// TIA Portal V16 export
// export: Created 2022-07-21T09:35:18.3308765Z, ExportSetting WithDefaults, DisplayName Totally Integrated Automation Portal, DisplayVersion V16 Update 4, DisplayName TIA Portal Version Control Interface, DisplayVersion V16 Update 2, DisplayName TIA Portal Openness, DisplayVersion V16 Update 4, DisplayName SINAMICS Startdrive Advanced, DisplayVersion V16 Update 5, DisplayName SINAMICS Startdrive G130, G150, S120, S150, SINAMICS MV, S210, DisplayVersion V16 Update 5, DisplayName SINAMICS Startdrive G110M, G120, G120C, G120D, G120P, G115D, DisplayVersion V16 Update 5, DisplayName STEP 7 Professional, DisplayVersion V16 Update 4, DisplayName STEP 7 Safety, DisplayVersion V16, DisplayName WinCC Advanced, DisplayVersion V16 Update 4
FUNCTION_BLOCK "fbATI"   // FB20, LAD
TITLE = ATI / Blok do obsługi ATI
{ S7_Optimized_Access := 'TRUE' }
VERSION : 0.1
// stored: AutoNumber false, IsIECCheckEnabled false, IsRetainMemResEnabled false, MemoryReserve 100, SetENOAutomatically false, UDAEnableTagReadback false
   VAR_INPUT
      portNr : UInt;   // numer portu / Port number
      generalRelease { ExternalWritable := 'False'} : Bool;   // Zezwolenie / General release
      autoEnable { ExternalWritable := 'False'} : Bool := true;   // Tryb automatyczny z HMI / Automatic mode from HMI
      ATI_ready { ExternalWritable := 'False'} : Bool;   // ATI -> PLC gotowe / ATI -> PLC ready
      ATI_passedTst { ExternalWritable := 'False'} : Bool;   // ATI -> PLC test ok
      ATI_failedTst { ExternalWritable := 'False'} : Bool;   // ATI -> PLC test nok
      ATI_fault { ExternalWritable := 'False'} : Bool;   // ATI -> PLC błąd / ATI -> PLC fault
      ATI_calMode { ExternalWritable := 'False'} : Bool;   // ATI -> PLC tryb kalibracji / ATI -> PLC calibration
      chuckClosed { ExternalWritable := 'False'} : Bool;   // Chuck zamknięty / Chuck closed
      partPlaced { ExternalWritable := 'False'} : Bool;   // Filtr w pozycji / Filter in position
      autoPenCal : Bool;   // Żądanie kalibracji / Calibration request
      group : "typeGroup";   // Grupa / Group
   END_VAR
   VAR_OUTPUT
      autoSelect { ExternalWritable := 'False'} : Bool;   // PLC -> ATI Tryb auto / PLC -> ATI Automatic mode
      extStart { ExternalWritable := 'False'} : Bool;   // PLC -> ATI Zewnętrzny start / PLC -> ATI External start
      penCal { ExternalWritable := 'False'} : Bool;   // PLC -> ATI Pen Cal
      ATIexists { ExternalWritable := 'False'} : Bool;   // ATI -> ext. ATI załączone z HMI / ATI -> ext. ATI on from HMI
      calIsRunning : Bool;   // kalibracja aktywna / calibration active
      calElapsedTime : Time;   // czas trwania kalibracji / calibration duration
      errorSendPort : Bool;   // Błąd bloku P2P Send / Block error P2P Send
      errorRecvPort : Bool;   // Błąd bloku P2P Receive / Block error P2P Receive
      errorCom : Bool;   // Błąd koumikacji : związany z Receive / Communication error : Receive related
   END_VAR
   VAR_IN_OUT
      ATI : "typeTester";   // Dane HMI / HMI data
      ATIP2P : "typeATIP2P";
      instRecvP2P : Receive_P2P;
      instSendP2P : Send_P2P;
   END_VAR
   VAR
      statTimerPenCalPls { ExternalWritable := 'False'; S7_SetPoint := 'True'} : TON_TIME;
      statTimerStartPls { ExternalWritable := 'False'; S7_SetPoint := 'True'} : TON_TIME;
      staRecvNDR { S7_SetPoint := 'True'} : Bool;
      statRecvError : Bool;
      statRecvStatus : Word;
      statRecvLength : UInt;
      statRecievedData : String;
      statSendData : String;
      statSendTrigger : Bool;
      statSendLength : UInt;
      statSendDone : Bool;
      statSendError : Bool;
      statSendStatus : Word;
      stat1Char : String;
      instDelaySendTG : TP_TIME;
      instDelayErrorRecvTG : TON_TIME;
      statWaitingForRecvTG : Bool;
      statDelayErrorProcess : Time;
      NewResultOKDigit { S7_SetPoint := 'True'} : Bool;
      NewResultOKDigit_RTIG : R_TRIG;
      NewResultNOKDigit : Bool;
      NewResultNOKDigit_RTIG : R_TRIG;
      sNegEdge : Array[0..7] of Bool;
      sPosEdge : Array[0..7] of Bool;
      sEqual : Bool;
   END_VAR
   VAR_TEMP
      tempCancelCalMode : Bool;   // Reset trybu kalibracji / Reset calibration mode
      tempAutoModeActive : Bool;   // Tryb auto/krokowy aktywny / Automatic/sequential mode active
      tempModeActive : Bool;   // Tryb aktywny / Active mode
      tempRetVal : Int;
      tempREQSend : Bool;
      tempCount : Int;
      tempVarTimeCAL : Time;
      tempCALerror : Bool;
      temp_cRL : Char;
      temp_sRL : String;
      tempStr : String;
      tempEqual : Bool;
      tempStatus3 : Bool;
   END_VAR
   VAR CONSTANT
      cTIME_OFF_SIGNAL : Time := T#1s;   // Czas opóźnienia dla alarmu 0 / delay alarm 0
      cTIME_ERR_PROCESS : Time := T#90s;
   END_VAR
   // // ATI.cmd.enable : Włączenie trybu automatycznego / Start automatic mode
   VAR_TEMP   // added for the SCL form of the ladder/FBD networks
      _w1 : Bool;
      _w2 : Bool;
   END_VAR
BEGIN

REGION Network 1: Alarm 1 - ATI fault / Alarm 1 - Błąd ATI
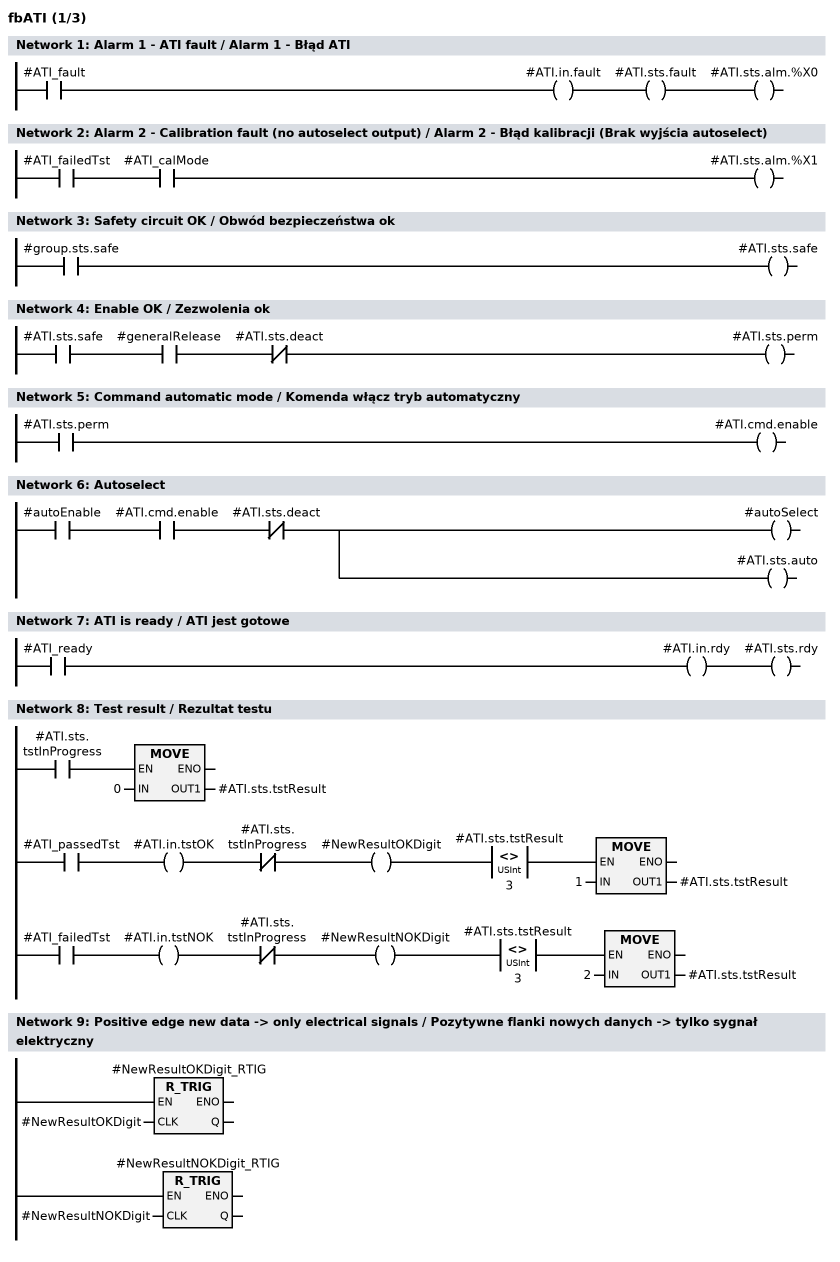
   RUNG wire#powerrail
      Contact( #ATI_fault )
      Coil( #ATI.in.fault )
      Coil( #ATI.sts.fault )
      Coil( #ATI.sts.alm.%X0 )
   END_RUNG
   // the same network as SCL:
   #ATI.in.fault := #ATI_fault;
   #ATI.sts.fault := #ATI_fault;
   #ATI.sts.alm.%X0 := #ATI_fault;
END_REGION

REGION Network 2: Alarm 2 - Calibration fault (no autoselect output) / Alarm 2 - Błąd kalibracji (Brak wyjścia autoselect)
   RUNG wire#powerrail
      Contact( #ATI_failedTst )
      Contact( #ATI_calMode )
      Coil( #ATI.sts.alm.%X1 )
   END_RUNG
   // the same network as SCL:
   #ATI.sts.alm.%X1 := #ATI_failedTst AND #ATI_calMode;
END_REGION

REGION Network 3: Safety circuit OK / Obwód bezpieczeństwa ok
   RUNG wire#powerrail
      Contact( #group.sts.safe )
      Coil( #ATI.sts.safe )
   END_RUNG
   // the same network as SCL:
   #ATI.sts.safe := #group.sts.safe;
END_REGION

REGION Network 4: Enable OK / Zezwolenia ok
   RUNG wire#powerrail
      Contact( #ATI.sts.safe )
      Contact( #generalRelease )
      I_Contact( #ATI.sts.deact )
      Coil( #ATI.sts.perm )
   END_RUNG
   // the same network as SCL:
   #ATI.sts.perm := #ATI.sts.safe AND #generalRelease AND NOT #ATI.sts.deact;
END_REGION

REGION Network 5: Command automatic mode / Komenda włącz tryb automatyczny
   RUNG wire#powerrail
      Contact( #ATI.sts.perm )
      Coil( #ATI.cmd.enable )
   END_RUNG
   // the same network as SCL:
   #ATI.cmd.enable := #ATI.sts.perm;
END_REGION

REGION Network 6: Autoselect
   RUNG wire#powerrail
      Contact( #autoEnable )
      Contact( #ATI.cmd.enable )
      I_Contact( #ATI.sts.deact )
      wire#w1
      Coil( #autoSelect )
   END_RUNG
   RUNG wire#w1
      Coil( #ATI.sts.auto )
   END_RUNG
   // the same network as SCL:
   #autoSelect := #autoEnable AND #ATI.cmd.enable AND NOT #ATI.sts.deact;
   #ATI.sts.auto := #autoSelect;
END_REGION

REGION Network 7: ATI is ready / ATI jest gotowe
   RUNG wire#powerrail
      Contact( #ATI_ready )
      Coil( #ATI.in.rdy )
      Coil( #ATI.sts.rdy )
   END_RUNG
   // the same network as SCL:
   #ATI.in.rdy := #ATI_ready;
   #ATI.sts.rdy := #ATI_ready;
END_REGION

REGION Network 8: Test result / Rezultat testu
   RUNG wire#powerrail
      Contact( #ATI.sts.tstInProgress )
      Move(in := 0, out1 => #ATI.sts.tstResult)
   END_RUNG
   RUNG wire#powerrail
      Contact( #ATI_passedTst )
      Coil( #ATI.in.tstOK )
      I_Contact( #ATI.sts.tstInProgress )
      Coil( #NewResultOKDigit )
      { S7_Templates := "SrcType := USInt" } NE_Contact(in1 := #ATI.sts.tstResult, in2 := 3)
      Move(in := 1, out1 => #ATI.sts.tstResult)
   END_RUNG
   RUNG wire#powerrail
      Contact( #ATI_failedTst )
      Coil( #ATI.in.tstNOK )
      I_Contact( #ATI.sts.tstInProgress )
      Coil( #NewResultNOKDigit )
      { S7_Templates := "SrcType := USInt" } NE_Contact(in1 := #ATI.sts.tstResult, in2 := 3)
      Move(in := 2, out1 => #ATI.sts.tstResult)
   END_RUNG
   // the same network as SCL:
   IF #ATI.sts.tstInProgress THEN #ATI.sts.tstResult := 0; END_IF;
   #ATI.in.tstOK := #ATI_passedTst;
   #NewResultOKDigit := #ATI_passedTst AND NOT #ATI.sts.tstInProgress;
   IF #NewResultOKDigit AND (#ATI.sts.tstResult <> 3) THEN #ATI.sts.tstResult := 1; END_IF;
   #ATI.in.tstNOK := #ATI_failedTst;
   #NewResultNOKDigit := #ATI_failedTst AND NOT #ATI.sts.tstInProgress;
   IF #NewResultNOKDigit AND (#ATI.sts.tstResult <> 3) THEN #ATI.sts.tstResult := 2; END_IF;
END_REGION

REGION Network 9: Positive edge new data -> only electrical signals / Pozytywne flanki nowych danych -> tylko sygnał elektryczny
   RUNG wire#powerrail
      #NewResultOKDigit_RTIG.R_TRIG(CLK := #NewResultOKDigit, Q =>)
   END_RUNG
   RUNG wire#powerrail
      #NewResultNOKDigit_RTIG.R_TRIG(CLK := #NewResultNOKDigit, Q =>)
   END_RUNG
   // the same network as SCL:
   #NewResultOKDigit_RTIG(CLK := #NewResultOKDigit);   // R_TRIG
   #NewResultNOKDigit_RTIG(CLK := #NewResultNOKDigit);   // R_TRIG
END_REGION

REGION Network 10: Alarm 4 - No RS232 data after test / Alarm 4 - Brak danych RS232 po teście
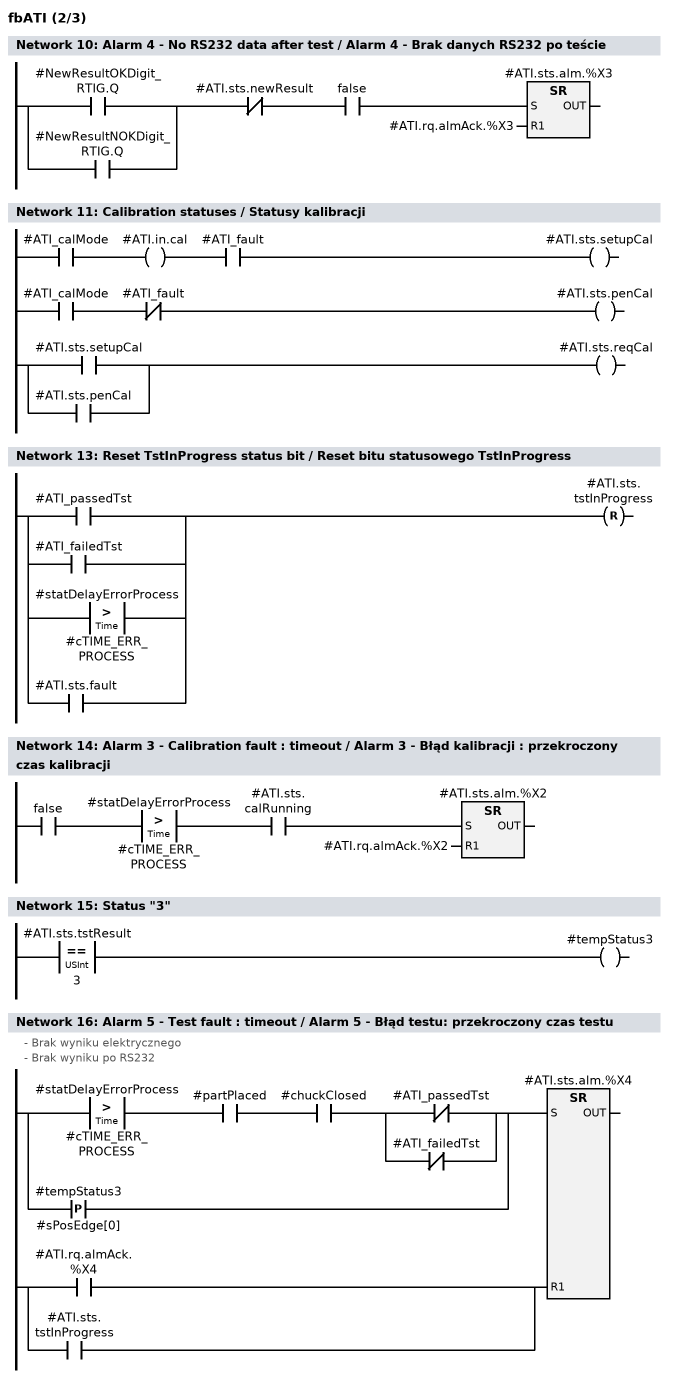
   RUNG wire#powerrail
      Contact( #NewResultOKDigit_RTIG.Q )
      wire#w1
      I_Contact( #ATI.sts.newResult )
      Contact( false )
      S_SR(operand := #ATI.sts.alm.%X3, r1 := #ATI.rq.almAck.%X3)
   END_RUNG
   RUNG wire#powerrail
      Contact( #NewResultNOKDigit_RTIG.Q )
   END_RUNG wire#w1
   // the same network as SCL:
   IF (#NewResultOKDigit_RTIG.Q OR #NewResultNOKDigit_RTIG.Q) AND NOT #ATI.sts.newResult AND false THEN
       #ATI.sts.alm.%X3 := TRUE;   // SR flip-flop
   END_IF;
   IF #ATI.rq.almAck.%X3 THEN #ATI.sts.alm.%X3 := FALSE; END_IF;
END_REGION

REGION Network 11: Calibration statuses / Statusy kalibracji
   RUNG wire#powerrail
      Contact( #ATI_calMode )
      Coil( #ATI.in.cal )
      Contact( #ATI_fault )
      Coil( #ATI.sts.setupCal )
   END_RUNG
   RUNG wire#powerrail
      Contact( #ATI_calMode )
      I_Contact( #ATI_fault )
      Coil( #ATI.sts.penCal )
   END_RUNG
   RUNG wire#powerrail
      Contact( #ATI.sts.setupCal )
      wire#w1
      Coil( #ATI.sts.reqCal )
   END_RUNG
   RUNG wire#powerrail
      Contact( #ATI.sts.penCal )
   END_RUNG wire#w1
   // the same network as SCL:
   #ATI.in.cal := #ATI_calMode;
   #ATI.sts.setupCal := #ATI_calMode AND #ATI_fault;
   #ATI.sts.penCal := #ATI_calMode AND NOT #ATI_fault;
   #ATI.sts.reqCal := #ATI.sts.setupCal OR #ATI.sts.penCal;
END_REGION

REGION Network 12 (SCL): ATI control / Sterowanie ATI

   #tempAutoModeActive := #group.sts.auto OR #group.sts.step;
   #tempModeActive := #tempAutoModeActive OR #group.sts.manual; //jakikolwiek tryb wybrany

   //Testy filtrów
   IF #ATI_ready AND NOT #ATI_fault THEN

       //start test filtra
       IF #autoSelect AND ((#tempAutoModeActive AND #partPlaced) OR (#group.sts.manual AND #ATI.rq.handStart))
           AND #chuckClosed AND NOT (#ATI_passedTst OR #ATI_failedTst) AND NOT #extStart THEN
           #extStart := TRUE;
           #ATI.sts.tstInProgress := TRUE;
       END_IF;

       //wymuszenie kalibracji podczas normalnej pracy
       IF #autoSelect AND #group.sts.manual AND NOT #partPlaced AND #chuckClosed AND #ATI.rq.rqPenCal AND NOT #penCal THEN
           #penCal := TRUE;
       END_IF;

   //Zadanie kalibracji
   ELSIF #ATI_calMode THEN

       //po starcie systemu (bład na ATI)
       IF #ATI.sts.setupCal THEN

           //tylko w trybie recznym ?
           IF #group.sts.manual AND #autoSelect AND NOT #partPlaced AND #chuckClosed AND #ATI.rq.startCal AND NOT #extStart THEN
               #extStart := TRUE;
               #ATI.sts.calRunning := TRUE;
           END_IF;

       //podczas normalnej pracy, po wcześniejszym jego wymuszeniu    
       ELSIF #ATI.sts.penCal THEN

           IF #tempModeActive AND #autoSelect AND NOT #partPlaced AND #chuckClosed AND (#ATI.rq.startCal OR #autoPenCal) AND NOT #extStart THEN
               #extStart := TRUE;
               #ATI.sts.calRunning := TRUE;
           END_IF;
       END_IF;
   END_IF;

   #statTimerStartPls(IN := #extStart,
                      PT := #cTIME_OFF_SIGNAL);
   #statTimerPenCalPls(IN := #penCal,
                       PT := #cTIME_OFF_SIGNAL);

   "fcCounterTime"(inEnableCount := true,
                   inReset := #extStart,
                   inValue := "CycleTimeData".PrevScanTime.Time,
                   ioCounter := #statDelayErrorProcess);

   IF #statTimerStartPls.Q THEN
       #extStart := FALSE;
   END_IF;

   IF #statTimerPenCalPls.Q THEN
       #penCal := FALSE;
   END_IF;

   IF #ATI.sts.calRunning THEN
       #calIsRunning := TRUE;
       #calElapsedTime := #statDelayErrorProcess;
   ELSE
       #calIsRunning := FALSE;
       #calElapsedTime := t#0ms;
   END_IF;
END_REGION

REGION Network 13: Reset TstInProgress status bit / Reset bitu statusowego TstInProgress
   RUNG wire#powerrail
      Contact( #ATI_passedTst )
      wire#w1
      R_Coil( #ATI.sts.tstInProgress )
   END_RUNG
   RUNG wire#powerrail
      Contact( #ATI_failedTst )
   END_RUNG wire#w1
   RUNG wire#powerrail
      { S7_Templates := "SrcType := Time" } GT_Contact(in1 := #statDelayErrorProcess, in2 := #cTIME_ERR_PROCESS)
   END_RUNG wire#w1
   RUNG wire#powerrail
      Contact( #ATI.sts.fault )
   END_RUNG wire#w1
   // the same network as SCL:
   IF #ATI_passedTst OR #ATI_failedTst OR (#statDelayErrorProcess > #cTIME_ERR_PROCESS) OR #ATI.sts.fault THEN
       #ATI.sts.tstInProgress := FALSE;
   END_IF;
END_REGION

REGION Network 14: Alarm 3 - Calibration fault : timeout / Alarm 3 - Błąd kalibracji : przekroczony czas kalibracji
   RUNG wire#powerrail
      Contact( false )
      { S7_Templates := "SrcType := Time" } GT_Contact(in1 := #statDelayErrorProcess, in2 := #cTIME_ERR_PROCESS)
      Contact( #ATI.sts.calRunning )
      S_SR(operand := #ATI.sts.alm.%X2, r1 := #ATI.rq.almAck.%X2)
   END_RUNG
   // the same network as SCL:
   IF false AND (#statDelayErrorProcess > #cTIME_ERR_PROCESS) AND #ATI.sts.calRunning THEN
       #ATI.sts.alm.%X2 := TRUE;   // SR flip-flop
   END_IF;
   IF #ATI.rq.almAck.%X2 THEN #ATI.sts.alm.%X2 := FALSE; END_IF;
END_REGION

REGION Network 15: Status "3"
   RUNG wire#powerrail
      { S7_Templates := "SrcType := USInt" } EQ_Contact(in1 := #ATI.sts.tstResult, in2 := 3)
      Coil( #tempStatus3 )
   END_RUNG
   // the same network as SCL:
   #tempStatus3 := #ATI.sts.tstResult = 3;
END_REGION

REGION Network 16: Alarm 5 - Test fault : timeout / Alarm 5 - Błąd testu: przekroczony czas testu
   // - Brak wyniku elektrycznego
   // - Brak wyniku po RS232
   RUNG wire#powerrail
      { S7_Templates := "SrcType := Time" } GT_Contact(in1 := #statDelayErrorProcess, in2 := #cTIME_ERR_PROCESS)
      Contact( #partPlaced )
      Contact( #chuckClosed )
      wire#w1
      I_Contact( #ATI_passedTst )
      wire#w2
      S_SR(operand := #ATI.sts.alm.%X4, r1 := wire#w3)
   END_RUNG
   RUNG wire#w1
      I_Contact( #ATI_failedTst )
   END_RUNG wire#w2
   RUNG wire#powerrail
      P_Contact(operand := #tempStatus3, bit := #sPosEdge[0])
   END_RUNG wire#w2
   RUNG wire#powerrail
      Contact( #ATI.rq.almAck.%X4 )
   END_RUNG wire#w3
   RUNG wire#powerrail
      Contact( #ATI.sts.tstInProgress )
   END_RUNG wire#w3
   // the same network as SCL:
   #_w1 := #tempStatus3 AND NOT #sPosEdge[0];   // rising edge of #tempStatus3
   #sPosEdge[0] := #tempStatus3;
   IF ((#statDelayErrorProcess > #cTIME_ERR_PROCESS) AND #partPlaced AND #chuckClosed AND (NOT #ATI_passedTst OR NOT #ATI_failedTst)) OR #_w1 THEN
       #ATI.sts.alm.%X4 := TRUE;   // SR flip-flop
   END_IF;
   IF #ATI.rq.almAck.%X4 OR #ATI.sts.tstInProgress THEN #ATI.sts.alm.%X4 := FALSE; END_IF;
END_REGION

REGION Network 17: Calibration in progress / Trwa proces kalibracji
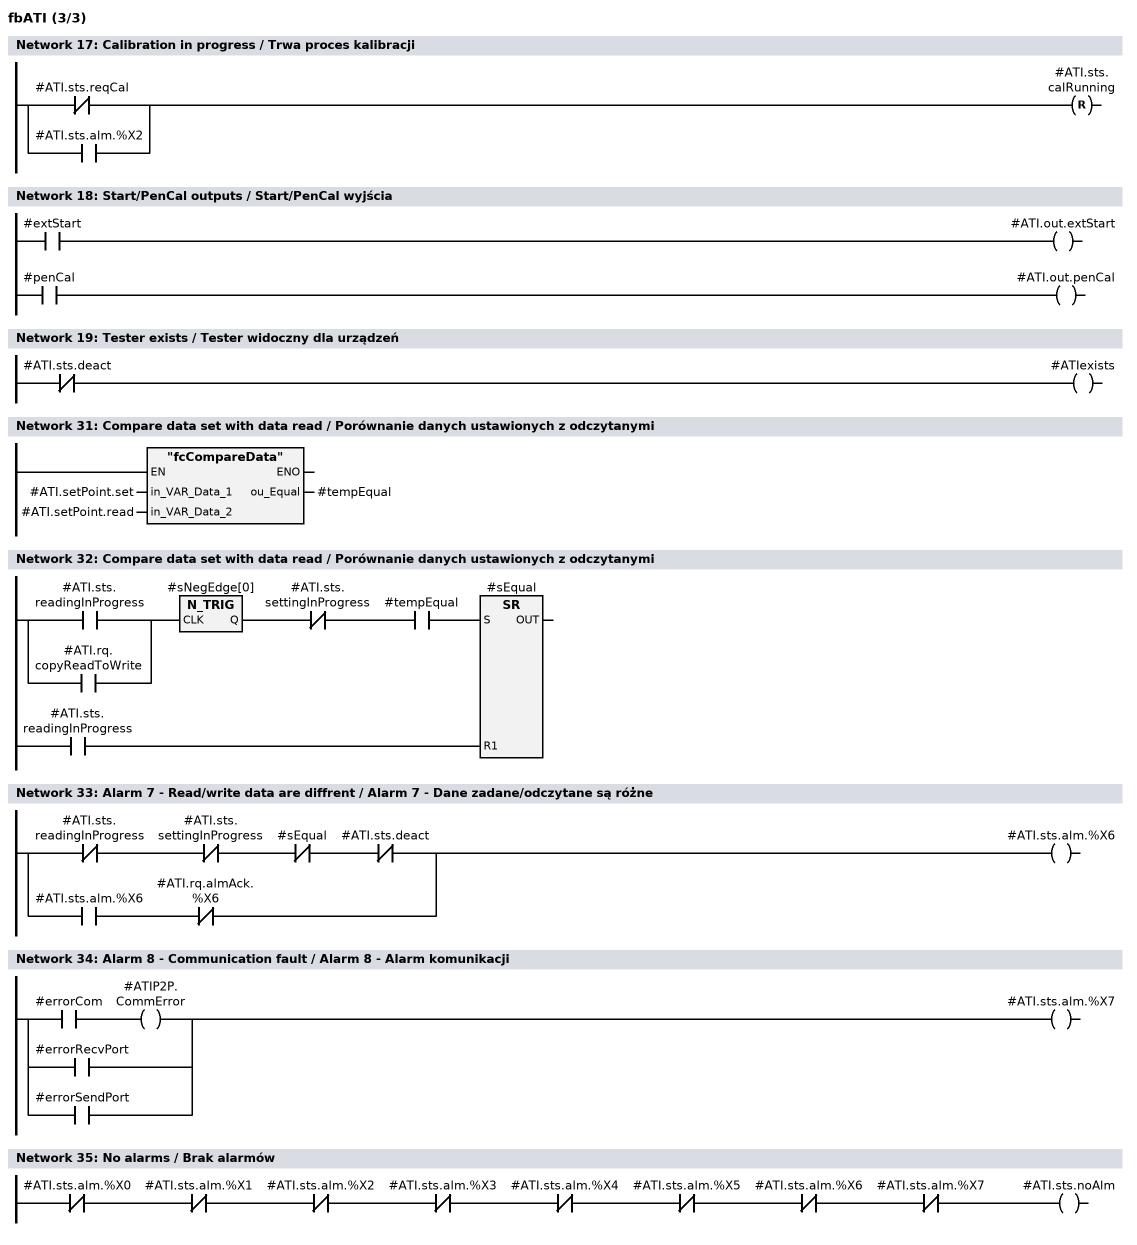
   RUNG wire#powerrail
      I_Contact( #ATI.sts.reqCal )
      wire#w1
      R_Coil( #ATI.sts.calRunning )
   END_RUNG
   RUNG wire#powerrail
      Contact( #ATI.sts.alm.%X2 )
   END_RUNG wire#w1
   // the same network as SCL:
   IF NOT #ATI.sts.reqCal OR #ATI.sts.alm.%X2 THEN #ATI.sts.calRunning := FALSE; END_IF;
END_REGION

REGION Network 18: Start/PenCal outputs / Start/PenCal wyjścia
   RUNG wire#powerrail
      Contact( #extStart )
      Coil( #ATI.out.extStart )
   END_RUNG
   RUNG wire#powerrail
      Contact( #penCal )
      Coil( #ATI.out.penCal )
   END_RUNG
   // the same network as SCL:
   #ATI.out.extStart := #extStart;
   #ATI.out.penCal := #penCal;
END_REGION

REGION Network 19: Tester exists / Tester widoczny dla urządzeń
   RUNG wire#powerrail
      I_Contact( #ATI.sts.deact )
      Coil( #ATIexists )
   END_RUNG
   // the same network as SCL:
   #ATIexists := NOT #ATI.sts.deact;
END_REGION

REGION Network 20 (SCL): ### FIFO buffer send telegram handling / ### Obsługa kolejnych telegramów do wysyłki z bufora FIFO

   (*
       IF #ATIP2P.CounterMsg < "ATI_MaxMsg" THEN
           #ATIP2P.BufferFull := FALSE;
       END_IF;

       IF #ATIP2P.CounterMsg > 0 THEN

           #statSendTrigger := TRUE;
           #statSendData := #ATIP2P.P2PSend[1].buffer;
           #statSendLength := INT_TO_UINT(LEN(#ATIP2P.P2PSend[1].buffer));

       ELSE
           #statSendTrigger := FALSE;
       END_IF;

   *)
END_REGION

REGION Network 21 (SCL): ### Ports handling / ### Obsługa portów
   (*
       #tempREQSend := #statSendTrigger //Trigger z bufora danych do wysyłyki
       AND NOT #instDelaySendTG.Q      //zwłoka czasowa pomiedzy kolejnymi telegramami
       AND NOT #statWaitingForRecvTG   //brak oczekiwania na telegram zwrotny
       AND NOT #errorCom;              //brak błędu komunikacji

       // Send data
       #instSendP2P(REQ := #tempREQSend,
                    "PORT" := #portNr,
                    BUFFER := #statSendData,
                    LENGTH := #statSendLength,
                    DONE => #statSendDone,
                    ERROR => #statSendError,
                    STATUS => #statSendStatus);

       // Read data
       #instRecvP2P("PORT" := #portNr,
                    BUFFER := #statRecievedData,
                    NDR => #staRecvNDR,
                    ERROR => #statRecvError,
                    STATUS => #statRecvStatus,
                    LENGTH => #statRecvLength);
   *)
END_REGION

REGION Network 22 (SCL): ### Telegram send/received / ### Telegram odebrany/wysłany

   (* REGION Kompletny telegram wysłany
       IF #statSendDone OR #statSendError THEN

           //zapamietanie ostatniego wyslanego telegramu
           #ATIP2P.LastSendMsg := #ATIP2P.P2PSend[1].buffer;

           //brak oczekiwania na telegram zwrotny
           IF NOT #ATIP2P.P2PSend[1].ReqRcvMsg THEN

               //przesuniecie kolejki FIFO i wysłanie nowego Msg
               #tempRetVal := MOVE_BLK_VARIANT(SRC := #ATIP2P.P2PSend,
                                               COUNT := INT_TO_UDINT("ATI_MaxMsg") - 1,
                                               SRC_INDEX := 1,
                                               DEST_INDEX := 0,
                                               DEST => #ATIP2P.P2PSend);

               "fcClearData"(io_VAR_Data := #ATIP2P.P2PSend[#ATIP2P.CounterMsg]);
               IF #ATIP2P.CounterMsg > 0 THEN
                   #ATIP2P.CounterMsg := #ATIP2P.CounterMsg - 1;
               END_IF;
           ELSE
               #statWaitingForRecvTG := TRUE;
           END_IF;

       END_IF;
   END_REGION

   REGION Telegram odebrany
       #ATIP2P.P2PRecv.newMsg := #staRecvNDR;
       #ATIP2P.P2PRecv.buffer := #statRecievedData;

       IF #staRecvNDR THEN
           #statWaitingForRecvTG := FALSE;

           //przesuniecie kolejki FIFO i wysłanie nowego Msg
           #tempRetVal := MOVE_BLK_VARIANT(SRC := #ATIP2P.P2PSend,
                                           COUNT := INT_TO_UDINT("ATI_MaxMsg")-1,
                                           SRC_INDEX := 1,
                                           DEST_INDEX := 0,
                                           DEST => #ATIP2P.P2PSend);

           "fcClearData"(io_VAR_Data := #ATIP2P.P2PSend[#ATIP2P.CounterMsg]);
           IF #ATIP2P.CounterMsg > 0 THEN
               #ATIP2P.CounterMsg := #ATIP2P.CounterMsg - 1;
           END_IF;
       END_IF;
   END_REGION *)
END_REGION

REGION Network 23 (SCL): ### Communication error / ### Błąd komunikacji

   (* REGION Obsługa błedu komunikacji
       #instDelayErrorRecvTG(IN := #statWaitingForRecvTG,
                             PT := t#5s);

       //Timeout na odpowiedz od ATI
       IF #instDelayErrorRecvTG.Q THEN
           #statWaitingForRecvTG := FALSE;
           #errorCom := TRUE;
       END_IF;

       //błędy kanalów P2P
       IF #statRecvError THEN
           #errorRecvPort := true;
       END_IF;

       IF #statSendError THEN
           #errorSendPort := true;
       END_IF;

       //reset błędów
       IF #ATI.rq.almAck.%X0 THEN
           #errorRecvPort := FALSE;
           #errorSendPort := FALSE;

           IF #errorCom THEN
               FOR #tempCount := 1 TO "ATI_MaxMsg" DO
                   "fcClearData"(io_VAR_Data := #ATIP2P.P2PSend[#tempCount]);
               END_FOR;

               #ATIP2P.CounterMsg := 0;
               #errorCom := FALSE;
           END_IF;

       END_IF;

   END_REGION *)
END_REGION

REGION Network 24 (SCL): ### Delay timer / ### Timer opóźniajacy

   (* // Opoznienie pomiedzy kolejnymi telegramami
   #instDelaySendTG(IN := #statSendDone OR #statSendError,
                    PT := t#1000ms); *)
END_REGION

REGION Network 25 (SCL): *** FIFO buffer send telegram handling / *** Obsługa kolejnych telegramów do wysyłki z bufora FIFO

   #temp_cRL := BYTE_TO_CHAR(16#D);
   #temp_sRL := CHAR_TO_STRING(IN := #temp_cRL);

    IF #ATIP2P.CounterMsg < "ATI_MaxMsg" THEN
       #ATIP2P.BufferFull := FALSE;
   END_IF;

   IF #ATIP2P.CounterMsg > 0 THEN

       IF NOT #statSendTrigger AND
           NOT #statWaitingForRecvTG AND   //brak oczekiwania na telegram zwrotny
           NOT #errorCom THEN              //brak błędu komunikacjiTHEN

           #statSendTrigger := TRUE;
           #statSendData := #ATIP2P.P2PSend[1].buffer;
           #statSendLength := INT_TO_UINT(LEN(#ATIP2P.P2PSend[1].buffer));
           #stat1Char := LEFT(IN := #statSendData, L := 1); //1 znak do wysyłki
           #statSendData := DELETE(IN := #statSendData, L := 1, P := 1); //usuniecie wysyłanego znaku

       END_IF;
   ELSE
       #statSendTrigger := FALSE;
   END_IF;
END_REGION

REGION Network 26 (SCL): *** Ports handling / *** Obsługa portów

   #tempREQSend := #statSendTrigger //Trigger z bufora danych do wysyłyki
   AND NOT #instDelaySendTG.Q      //zwłoka czasowa pomiedzy kolejnymi telegramami
   AND NOT #statWaitingForRecvTG   //brak oczekiwania na telegram zwrotny
   AND NOT #errorCom;               //brak błędu komunikacji

   // Send data
   #instSendP2P(REQ := #tempREQSend,
                PORT := #portNr,
                BUFFER := #stat1Char,
                LENGTH := 1,
                DONE => #statSendDone,
                ERROR => #statSendError,
                STATUS => #statSendStatus);

   // Read data
   #instRecvP2P(PORT := #portNr,
                BUFFER := #statRecievedData,
                NDR => #staRecvNDR,
                ERROR => #statRecvError,
                STATUS => #statRecvStatus,
                LENGTH => #statRecvLength);
END_REGION

REGION Network 27 (SCL): *** Telegram send/received / *** Telegram odebrany/wysłany

   REGION Kompletny telegram wysłany
       IF (#statSendDone AND #stat1Char = #temp_sRL) OR #statSendError THEN

           //zapamietanie ostatniego wyslanego telegramu
           #ATIP2P.LastSendMsg := #ATIP2P.P2PSend[1].buffer;
           #statSendTrigger := FALSE;

           //brak oczekiwania na telegram zwrotny
           IF NOT #ATIP2P.P2PSend[1].ReqRcvMsg THEN

               //przesuniecie kolejki FIFO i wysłanie nowego Msg
               #tempRetVal := MOVE_BLK_VARIANT(SRC := #ATIP2P.P2PSend,
                                               COUNT := INT_TO_UDINT("ATI_MaxMsg") - 1,
                                               SRC_INDEX := 1,
                                               DEST_INDEX := 0,
                                               DEST => #ATIP2P.P2PSend);

               "fcClearData"(io_VAR_Data := #ATIP2P.P2PSend[#ATIP2P.CounterMsg]);
               IF #ATIP2P.CounterMsg > 0 THEN
                   #ATIP2P.CounterMsg := #ATIP2P.CounterMsg - 1;
               END_IF;
           ELSE
               #statWaitingForRecvTG := TRUE;
           END_IF;

       END_IF;
   END_REGION

   REGION Telegram odebrany
       #ATIP2P.P2PRecv.newMsg := #staRecvNDR;
       #ATIP2P.P2PRecv.buffer := #statRecievedData;

       IF #staRecvNDR THEN
           #statWaitingForRecvTG := FALSE;

           //przesuniecie kolejki FIFO i wysłanie nowego Msg
           #tempRetVal := MOVE_BLK_VARIANT(SRC := #ATIP2P.P2PSend,
                                           COUNT := INT_TO_UDINT("ATI_MaxMsg")-1,
                                           SRC_INDEX := 1,
                                           DEST_INDEX := 0,
                                           DEST => #ATIP2P.P2PSend);

           "fcClearData"(io_VAR_Data := #ATIP2P.P2PSend[#ATIP2P.CounterMsg]);
           IF #ATIP2P.CounterMsg > 0 THEN
               #ATIP2P.CounterMsg := #ATIP2P.CounterMsg - 1;
           END_IF;
       END_IF;
   END_REGION
END_REGION

REGION Network 28 (SCL): *** Communication error / *** Błąd komunikacji

   REGION Obsługa błedu komunikacji
       #instDelayErrorRecvTG(IN := #statWaitingForRecvTG,
                             PT := t#5s);

       //Timeout na odpowiedz od ATI
       IF #instDelayErrorRecvTG.Q THEN
           #statWaitingForRecvTG := FALSE;
           #errorCom := TRUE;
       END_IF;

       //błędy kanalów P2P
       IF #statRecvError THEN
           #errorRecvPort := true;
       END_IF;

       IF #statSendError THEN
           #errorSendPort := true;
       END_IF;

       //reset błędów
       IF #ATI.rq.almAck.%X0 THEN
           #errorRecvPort := FALSE;
           #errorSendPort := FALSE;

           IF #errorCom THEN
               FOR #tempCount := 1 TO "ATI_MaxMsg" DO
                   "fcClearData"(io_VAR_Data := #ATIP2P.P2PSend[#tempCount]);
               END_FOR;

               #ATIP2P.CounterMsg := 0;
               #errorCom := FALSE;
           END_IF;

       END_IF;

   END_REGION
END_REGION

REGION Network 29 (SCL): *** Telegram char by char / *** Ustawianie telegramu (znak po znaku)

    IF (#statSendDone AND #stat1Char <> #temp_sRL) AND NOT #instDelaySendTG.Q THEN
       #stat1Char := LEFT(IN := #statSendData, L := 1); //1 znak do wysyłki
       #statSendData := DELETE(IN := #statSendData, L := 1, P := 1); //usuniecie wysyłanego znaku    
   END_IF;
END_REGION

REGION Network 30 (SCL): *** Delay timer / *** Timer opóźniajacy

   // Opoznienie pomiedzy kolejnymi telegramami
   #instDelaySendTG(IN := #statSendDone OR #statSendError,
                    PT := t#100ms);
END_REGION

REGION Network 31: Compare data set with data read / Porównanie danych ustawionych z odczytanymi
   RUNG wire#powerrail
      "fcCompareData"(in_VAR_Data_1 := #ATI.setPoint.set, in_VAR_Data_2 := #ATI.setPoint.read, ou_Equal => #tempEqual)
   END_RUNG
   // the same network as SCL:
   "fcCompareData"(in_VAR_Data_1 := #ATI.setPoint.set,
                   in_VAR_Data_2 := #ATI.setPoint.read,
                   ou_Equal => #tempEqual);
END_REGION

REGION Network 32: Compare data set with data read / Porównanie danych ustawionych z odczytanymi
   RUNG wire#powerrail
      Contact( #ATI.sts.readingInProgress )
      wire#w1
      N_Trig( #sNegEdge[0] )
      I_Contact( #ATI.sts.settingInProgress )
      Contact( #tempEqual )
      S_SR(operand := #sEqual, r1 := wire#w2)
   END_RUNG
   RUNG wire#powerrail
      Contact( #ATI.rq.copyReadToWrite )
   END_RUNG wire#w1
   RUNG wire#powerrail
      Contact( #ATI.sts.readingInProgress )
   END_RUNG wire#w2
   // the same network as SCL:
   #_w1 := #ATI.sts.readingInProgress OR #ATI.rq.copyReadToWrite;
   #_w2 := NOT #_w1 AND #sNegEdge[0];   // falling edge
   #sNegEdge[0] := #_w1;
   IF #_w2 AND NOT #ATI.sts.settingInProgress AND #tempEqual THEN
       #sEqual := TRUE;   // SR flip-flop
   END_IF;
   IF #ATI.sts.readingInProgress THEN #sEqual := FALSE; END_IF;
END_REGION

REGION Network 33: Alarm 7 - Read/write data are diffrent / Alarm 7 - Dane zadane/odczytane są różne
   RUNG wire#powerrail
      I_Contact( #ATI.sts.readingInProgress )
      I_Contact( #ATI.sts.settingInProgress )
      I_Contact( #sEqual )
      I_Contact( #ATI.sts.deact )
      wire#w1
      Coil( #ATI.sts.alm.%X6 )
   END_RUNG
   RUNG wire#powerrail
      Contact( #ATI.sts.alm.%X6 )
      I_Contact( #ATI.rq.almAck.%X6 )
   END_RUNG wire#w1
   // the same network as SCL:
   #ATI.sts.alm.%X6 := (NOT #ATI.sts.readingInProgress AND NOT #ATI.sts.settingInProgress AND NOT #sEqual AND NOT #ATI.sts.deact) OR (#ATI.sts.alm.%X6 AND NOT #ATI.rq.almAck.%X6);
END_REGION

REGION Network 34: Alarm 8 - Communication fault / Alarm 8 - Alarm komunikacji
   RUNG wire#powerrail
      Contact( #errorCom )
      Coil( #ATIP2P.CommError )
      wire#w1
      Coil( #ATI.sts.alm.%X7 )
   END_RUNG
   RUNG wire#powerrail
      Contact( #errorRecvPort )
   END_RUNG wire#w1
   RUNG wire#powerrail
      Contact( #errorSendPort )
   END_RUNG wire#w1
   // the same network as SCL:
   #ATIP2P.CommError := #errorCom;
   #ATI.sts.alm.%X7 := #errorCom OR #errorRecvPort OR #errorSendPort;
END_REGION

REGION Network 35: No alarms / Brak alarmów
   RUNG wire#powerrail
      I_Contact( #ATI.sts.alm.%X0 )
      I_Contact( #ATI.sts.alm.%X1 )
      I_Contact( #ATI.sts.alm.%X2 )
      I_Contact( #ATI.sts.alm.%X3 )
      I_Contact( #ATI.sts.alm.%X4 )
      I_Contact( #ATI.sts.alm.%X5 )
      I_Contact( #ATI.sts.alm.%X6 )
      I_Contact( #ATI.sts.alm.%X7 )
      Coil( #ATI.sts.noAlm )
   END_RUNG
   // the same network as SCL:
   #ATI.sts.noAlm := NOT #ATI.sts.alm.%X0 AND NOT #ATI.sts.alm.%X1 AND NOT #ATI.sts.alm.%X2 AND NOT #ATI.sts.alm.%X3 AND NOT #ATI.sts.alm.%X4 AND NOT #ATI.sts.alm.%X5 AND NOT #ATI.sts.alm.%X6 AND NOT #ATI.sts.alm.%X7;
END_REGION
END_FUNCTION_BLOCK
